FUNCTION F_PosUnderUpperBound : BOOL
VAR_INPUT
    fPosition: LREAL;
    stPositionState: ST_PositionState;
END_VAR


F_PosUnderUpperBound := fPosition < (stPositionState.fPosition + ABS(stPositionState.fDelta));

END_FUNCTION

(* stored: Version 1.1.0.1
   POU F_PosUnderUpperBound: Id {b5ee37fa-13c6-40f2-a7c7-9ac80833d78f}, SpecialFunc None *)
